Fanuc KAREL source: kt00116.KL

-- PROVISIONAL review KL for V770-1; original PC SHA256 bb3b05cc6ebd068e9e2a1367dbb604858096aad25b7d4729e2f2f28b6006a1c5
-- Incomplete behavior may be omitted. Consult companion uncertainty JSON. Do not deploy.
PROGRAM KT00116
%NOLOCKGROUP
VAR
  R2 : REAL
  OUT : REAL
-- UNRESOLVED_DECL Y1 type=002018
BEGIN
  -- UNRESOLVED_PC offsets 5-19; opcodes 2E,22,9D,33,B2
  -- UNRESOLVED_PC offsets 24-35; opcodes 2E,23
  -- UNRESOLVED_PC offsets 40-65; opcodes 22,9D,33,B1,21,29,64,29,6C,23
  -- UNRESOLVED_PC offsets 70-74; opcodes 7F
END KT00116
